{attribute 'OPC.UA.DA.StructuredType' := '1'}
TYPE ST_ResetError :
STRUCT
	bResetError		: BOOL; //true to reset error
	bResetWarning 	: BOOL; //true to reset warning
END_STRUCT
END_TYPE

(* stored: Version 1.1.0.1, ProductVersion 3.1.4024.9
   DUT ST_ResetError: Id {e9ba34a8-10cb-42af-81b1-35a6177abc71} *)
